// TIA Portal V20 export
TYPE "typeCmControlNode"
// stored: Namespace Unit1.Em6
   STRUCT
      interlock : "Unit1.Em6.typeCmControlNodeInterlock";
   END_STRUCT;
END_TYPE
